//     Box 64 (AT5100-0100)/DRV Controlword/Controlword <-> Data Pointer/Control
//     Box 64 (AT5100-0100)/DRV Statusword/Statusword <-> Data Pointer/Status
//     Box 64 (AT5100-0100)/DRV Target torque/Target torque <-> Data Pointer/Torque
//     Box 64 (AT5100-0100)/DRV Torque actual value/Torque actual value <-> Data Pointer/ActTorque
//     Box 64 (AT5100-0100)/XFB Inputs/Data <-> Data Pointer/HallSensorValues
//   (this object) <-> TcCOM Objects/XTS ProcessingUnit 1/XL Part 2/XL Module 53
//     Box 65 (AT5100-0100)/DRV Commutation angle/Commutation angle <-> Data Pointer/CommutationAngle
//     Box 65 (AT5100-0100)/DRV Controlword/Controlword <-> Data Pointer/Control
//     Box 65 (AT5100-0100)/DRV Statusword/Statusword <-> Data Pointer/Status
//     Box 65 (AT5100-0100)/DRV Target torque/Target torque <-> Data Pointer/Torque
//     Box 65 (AT5100-0100)/DRV Torque actual value/Torque actual value <-> Data Pointer/ActTorque
//     Box 65 (AT5100-0100)/XFB Inputs/Data <-> Data Pointer/HallSensorValues
//   (this object) <-> TcCOM Objects/XTS ProcessingUnit 1/XL Part 2/XL Module 54
//     Box 66 (AT5100-0100)/DRV Commutation angle/Commutation angle <-> Data Pointer/CommutationAngle
//     Box 66 (AT5100-0100)/DRV Controlword/Controlword <-> Data Pointer/Control
//     Box 66 (AT5100-0100)/DRV Statusword/Statusword <-> Data Pointer/Status
//     Box 66 (AT5100-0100)/DRV Target torque/Target torque <-> Data Pointer/Torque
//     Box 66 (AT5100-0100)/DRV Torque actual value/Torque actual value <-> Data Pointer/ActTorque
//     Box 66 (AT5100-0100)/XFB Inputs/Data <-> Data Pointer/HallSensorValues
//   (this object) <-> TcCOM Objects/XTS ProcessingUnit 1/XL Part 2/XL Module 55
//     Box 67 (AT5100-0100)/DRV Commutation angle/Commutation angle <-> Data Pointer/CommutationAngle
//     Box 67 (AT5100-0100)/DRV Controlword/Controlword <-> Data Pointer/Control
//     Box 67 (AT5100-0100)/DRV Statusword/Statusword <-> Data Pointer/Status
//     Box 67 (AT5100-0100)/DRV Target torque/Target torque <-> Data Pointer/Torque
//     Box 67 (AT5100-0100)/DRV Torque actual value/Torque actual value <-> Data Pointer/ActTorque
//     Box 67 (AT5100-0100)/XFB Inputs/Data <-> Data Pointer/HallSensorValues
//   (this object) <-> TcCOM Objects/XTS ProcessingUnit 1/XL Part 2/XL Module 56
//     Box 68 (AT5100-0100)/DRV Commutation angle/Commutation angle <-> Data Pointer/CommutationAngle
//     Box 68 (AT5100-0100)/DRV Controlword/Controlword <-> Data Pointer/Control
//     Box 68 (AT5100-0100)/DRV Statusword/Statusword <-> Data Pointer/Status
//     Box 68 (AT5100-0100)/DRV Target torque/Target torque <-> Data Pointer/Torque
//     Box 68 (AT5100-0100)/DRV Torque actual value/Torque actual value <-> Data Pointer/ActTorque
//     Box 68 (AT5100-0100)/XFB Inputs/Data <-> Data Pointer/HallSensorValues
//   (this object) <-> TcCOM Objects/XTS ProcessingUnit 1/XL Part 2/XL Module 57
//     Box 69 (AT5100-0100)/DRV Commutation angle/Commutation angle <-> Data Pointer/CommutationAngle
//     Box 69 (AT5100-0100)/DRV Controlword/Controlword <-> Data Pointer/Control
//     Box 69 (AT5100-0100)/DRV Statusword/Statusword <-> Data Pointer/Status
//     Box 69 (AT5100-0100)/DRV Target torque/Target torque <-> Data Pointer/Torque
//     Box 69 (AT5100-0100)/DRV Torque actual value/Torque actual value <-> Data Pointer/ActTorque
//     Box 69 (AT5100-0100)/XFB Inputs/Data <-> Data Pointer/HallSensorValues
//   (this object) <-> TcCOM Objects/XTS ProcessingUnit 1/XL Part 3/XL Module 1
//     Box 74 (AT5100-0100)/DRV Commutation angle/Commutation angle <-> Data Pointer/CommutationAngle
//     Box 74 (AT5100-0100)/DRV Controlword/Controlword <-> Data Pointer/Control
//     Box 74 (AT5100-0100)/DRV Statusword/Statusword <-> Data Pointer/Status
//     Box 74 (AT5100-0100)/DRV Target torque/Target torque <-> Data Pointer/Torque
//     Box 74 (AT5100-0100)/DRV Torque actual value/Torque actual value <-> Data Pointer/ActTorque
//     Box 74 (AT5100-0100)/XFB Inputs/Data <-> Data Pointer/HallSensorValues
//   (this object) <-> TcCOM Objects/XTS ProcessingUnit 1/XL Part 3/XL Module 2
//     Box 75 (AT5100-0100)/DRV Commutation angle/Commutation angle <-> Data Pointer/CommutationAngle
//     Box 75 (AT5100-0100)/DRV Controlword/Controlword <-> Data Pointer/Control
//     Box 75 (AT5100-0100)/DRV Statusword/Statusword <-> Data Pointer/Status
//     Box 75 (AT5100-0100)/DRV Target torque/Target torque <-> Data Pointer/Torque
//     Box 75 (AT5100-0100)/DRV Torque actual value/Torque actual value <-> Data Pointer/ActTorque
//     Box 75 (AT5100-0100)/XFB Inputs/Data <-> Data Pointer/HallSensorValues
//   (this object) <-> TcCOM Objects/XTS ProcessingUnit 1/XL Part 3/XL Module 3
//     Box 76 (AT5100-0100)/DRV Commutation angle/Commutation angle <-> Data Pointer/CommutationAngle
//     Box 76 (AT5100-0100)/DRV Controlword/Controlword <-> Data Pointer/Control
//     Box 76 (AT5100-0100)/DRV Statusword/Statusword <-> Data Pointer/Status
//     Box 76 (AT5100-0100)/DRV Target torque/Target torque <-> Data Pointer/Torque
//     Box 76 (AT5100-0100)/DRV Torque actual value/Torque actual value <-> Data Pointer/ActTorque
//     Box 76 (AT5100-0100)/XFB Inputs/Data <-> Data Pointer/HallSensorValues
//   (this object) <-> TcCOM Objects/XTS ProcessingUnit 1/XL Part 3/XL Module 4
//     Box 77 (AT5100-0100)/DRV Commutation angle/Commutation angle <-> Data Pointer/CommutationAngle
//     Box 77 (AT5100-0100)/DRV Controlword/Controlword <-> Data Pointer/Control
//     Box 77 (AT5100-0100)/DRV Statusword/Statusword <-> Data Pointer/Status
//     Box 77 (AT5100-0100)/DRV Target torque/Target torque <-> Data Pointer/Torque
//     Box 77 (AT5100-0100)/DRV Torque actual value/Torque actual value <-> Data Pointer/ActTorque
//     Box 77 (AT5100-0100)/XFB Inputs/Data <-> Data Pointer/HallSensorValues
//   (this object) <-> TcCOM Objects/XTS ProcessingUnit 1/XL Part 3/XL Module 46
//     Box 72 (AT5100-0100)/DRV Commutation angle/Commutation angle <-> Data Pointer/CommutationAngle
//     Box 72 (AT5100-0100)/DRV Controlword/Controlword <-> Data Pointer/Control
//     Box 72 (AT5100-0100)/DRV Statusword/Statusword <-> Data Pointer/Status
//     Box 72 (AT5100-0100)/DRV Target torque/Target torque <-> Data Pointer/Torque
//     Box 72 (AT5100-0100)/DRV Torque actual value/Torque actual value <-> Data Pointer/ActTorque
//     Box 72 (AT5100-0100)/XFB Inputs/Data <-> Data Pointer/HallSensorValues
//   (this object) <-> TcCOM Objects/XTS ProcessingUnit 1/XL Part 3/XL Module 47
//     Box 73 (AT5100-0100)/DRV Commutation angle/Commutation angle <-> Data Pointer/CommutationAngle
//     Box 73 (AT5100-0100)/DRV Controlword/Controlword <-> Data Pointer/Control
//     Box 73 (AT5100-0100)/DRV Statusword/Statusword <-> Data Pointer/Status
//     Box 73 (AT5100-0100)/DRV Target torque/Target torque <-> Data Pointer/Torque
//     Box 73 (AT5100-0100)/DRV Torque actual value/Torque actual value <-> Data Pointer/ActTorque
//     Box 73 (AT5100-0100)/XFB Inputs/Data <-> Data Pointer/HallSensorValues
//   (this object) <-> TcCOM Objects/XTS ProcessingUnit 1/XL Part 3/XL Module 5
//     Box 78 (AT5100-0100)/DRV Commutation angle/Commutation angle <-> Data Pointer/CommutationAngle
//     Box 78 (AT5100-0100)/DRV Controlword/Controlword <-> Data Pointer/Control
//     Box 78 (AT5100-0100)/DRV Statusword/Statusword <-> Data Pointer/Status
//     Box 78 (AT5100-0100)/DRV Target torque/Target torque <-> Data Pointer/Torque
//     Box 78 (AT5100-0100)/DRV Torque actual value/Torque actual value <-> Data Pointer/ActTorque
//     Box 78 (AT5100-0100)/XFB Inputs/Data <-> Data Pointer/HallSensorValues
//   (this object) <-> TcCOM Objects/XTS ProcessingUnit 1/XL Part 3/XL Module 6
//     Box 79 (AT5100-0100)/DRV Commutation angle/Commutation angle <-> Data Pointer/CommutationAngle
//     Box 79 (AT5100-0100)/DRV Controlword/Controlword <-> Data Pointer/Control
//     Box 79 (AT5100-0100)/DRV Statusword/Statusword <-> Data Pointer/Status
//     Box 79 (AT5100-0100)/DRV Target torque/Target torque <-> Data Pointer/Torque
//     Box 79 (AT5100-0100)/DRV Torque actual value/Torque actual value <-> Data Pointer/ActTorque
//     Box 79 (AT5100-0100)/XFB Inputs/Data <-> Data Pointer/HallSensorValues
//   (this object) <-> TcCOM Objects/XTS ProcessingUnit 1/XL Part 3/XL Module 7
//     Box 80 (AT5100-0100)/DRV Commutation angle/Commutation angle <-> Data Pointer/CommutationAngle
//     Box 80 (AT5100-0100)/DRV Controlword/Controlword <-> Data Pointer/Control
//     Box 80 (AT5100-0100)/DRV Statusword/Statusword <-> Data Pointer/Status
//     Box 80 (AT5100-0100)/DRV Target torque/Target torque <-> Data Pointer/Torque
//     Box 80 (AT5100-0100)/DRV Torque actual value/Torque actual value <-> Data Pointer/ActTorque
//     Box 80 (AT5100-0100)/XFB Inputs/Data <-> Data Pointer/HallSensorValues
//   (this object) <-> TcCOM Objects/XTS ProcessingUnit 1/XL Part 3/XL Module 8
//     Box 81 (AT5100-0100)/DRV Commutation angle/Commutation angle <-> Data Pointer/CommutationAngle
//     Box 81 (AT5100-0100)/DRV Controlword/Controlword <-> Data Pointer/Control
//     Box 81 (AT5100-0100)/DRV Statusword/Statusword <-> Data Pointer/Status
//     Box 81 (AT5100-0100)/DRV Target torque/Target torque <-> Data Pointer/Torque
//     Box 81 (AT5100-0100)/DRV Torque actual value/Torque actual value <-> Data Pointer/ActTorque
//     Box 81 (AT5100-0100)/XFB Inputs/Data <-> Data Pointer/HallSensorValues

CONFIGURATION PlanarTrackMovement_1
    RESOURCE PLC ON TwinCAT3
        TASK PlcTask(INTERVAL := T#1ms, PRIORITY := 20);
        PROGRAM MAIN WITH PlcTask : MAIN;
    END_RESOURCE
END_CONFIGURATION

// ---- GVLs/GVL_General.TcGVL
VAR_GLOBAL CONSTANT

	nNumMaxMovers : UDINT :=16;
	nNumMaxTracks : UDINT :=3;
 	fMagnetEntry : LREAL := 8750; //PLEASE ENTER THE MAGNET ENTRY!!!
	fMagnetExit : LREAL := 9450; //PLEASE ENTER THE MAGNET EXIT!!!
END_VAR

VAR_GLOBAL
	aStopPositions : ARRAY [1..nNumMaxMovers] OF LREAL;// := [2400, 1700, 1000, 300];
	XtsOutterLoopOid: OTCID := 16#1010480;	
	XtsShortcutOid: OTCID := 16#1010490;
END_VAR

VAR_GLOBAL PERSISTENT
	nNumMovers: UDINT := 4;
END_VAR

// ---- POUs/MAIN.TcPOU
PROGRAM MAIN
VAR
		
	bAllDone		: BOOL;
	bStopSequence	: BOOL;
	
	nCase 		: INT;
	nMoveState		: ARRAY[1..nNumMaxMovers] OF INT;
	
	aDynamics	: ARRAY[1..nNumMaxMovers] OF DynamicConstraint_PathXY;
	aDynamicsFast	: ARRAY[1..nNumMaxMovers] OF DynamicConstraint_PathXY;
	aMoveOnTrackOptions : ARRAY[1..20] OF ST_MoveOnTrackOptions;
	
	fbXtsEnvironment: FB_TcIoXtsEnvironment;
	
	nForCounter: UDINT;
	M,N,T,Tr : UDINT;
	dynamics: INT;
	
	// Magnet
	MagnetValue AT%Q*: INT;
	bMagnetOn : BOOL;	
	stPositionInfo: ST_PositionInfo;
		
	pwm: FB_PWM;
	
	IsMoverCommandedInShortcut: BOOL;
	IsMoverInBlockingArea: BOOL;
	nActStopPos: UINT := 1;
	Fp_error : R_Trig;
	Velo : LREAL := 500;
	Switch : BOOL;
	WithoutSwitch : BOOL := TRUE;
	SwtichOnly: BOOL;
	
	MoverStop 	AT%I* :BOOL;
	MoverStopDone AT%Q*		: BOOL;
	Info 		AT%Q*: BOOL;
	Operating	AT%Q*: BOOL;
	Process		AT%Q*: BOOL;
	Fault		AT%Q*: BOOL;
	Emergency	AT%Q*: BOOL;
	
	Voltage1 AT%I*: UDINT;
	Voltage2 AT%I*: UDINT;
	
	
	TcRestart : TC_Restart;
	Restart : BOOL;
	busy : BOOL;
	fp_start : R_Trig;
	bStartSequence: BOOL;
	
	FP_Counter : r_trig;
	Switchcounter : DINT;
	SwitchCurrent: INT :=12000; 
	test : LREAL;
	Horntimer : tp; 
	R_trigHorn : R_trig;
	
	TestPowerMat : BOOL;
	StopPos : LREAL := 7611;
	StopTime : TIME := T#8S;
	StopTimer :ARRAY[1..nNumMaxMovers] OF ton;
	StartTimer :ARRAY[1..nNumMaxMovers] OF BOOL;
	
	
	MoverPos :ARRAY[1..nNumMaxMovers] OF PositionXYC;
	ArcLength :ARRAY[1..nNumMaxMovers] OF LREAL;
	TrackPos :ARRAY[1..nNumMaxMovers] OF ARRAY[1..nNumMaxTracks] OF PositionXYC;
	
	GetMoverOnTrack : ReadTcCom;
	aMoverTrack : ARRAY[1..nNumMaxMovers] OF otcid;
	FirstMoverTrackPos : LREAL;
	MoverGap : LREAL;
	FTrigTrackCount : F_Trig;
	MoverNo  : UDINT;
END_VAR

fbXtsEnvironment.Init(TRUE);

Emergency :=  MoverStop;

Operating := NOT  MoverStop;
R_trigHorn(clk := Voltage1> 10000 OR Voltage2 >10000);
Horntimer(in:= ( R_trigHorn.Q ) , PT:= T#2S,Q=> info);

IF nCASE > 90 THEN
	Process := TRUE;
ELSE 
	Process := FALSE;	
END_IF





IF NOT fbXtsEnvironment.P_IsInitialized THEN
	RETURN;
END_IF





IF GetMoverOnTrack.GetComObject(MC_Tracks[1].MCTOPLC_STD.TrackOID)THEN
	aMoverTrack:= GetMoverOnTrack.GetValue();
END_IF







IF NOT MoverStop AND NOT MoverStopDone THEN
	FOR nForCounter:=1 TO nNumMovers DO
		aDynamics[nForCounter].SetValuesVADJ(8000, 8000, 8000, 20000);
		nCase := 140;
		//fbPlanarMover[nForCounter].McPlanarMover.Halt(MoverFeedback[nForCounter], aDynamics[nForCounter]);
	END_FOR		
	MoverStopDone := TRUE;
ELSIF 	MoverStop THEN
	MoverStopDone := FALSE;
END_IF


	TcRestart(
	NETID:= '', 
	RESTART:= Restart, 
	TMOUT:=T#5S , 
	BUSY=>busy , 
	ERR=> , 
	ERRID=> );


fp_start(clk:=bStartSequence);
IF fp_start.Q THEN
	nCase := 10;
	bStartSequence := FALSE;
END_IF



IsMoverInBlockingArea := FALSE;
FOR M := 1 TO nNumMovers DO///Movers
	StopTimer[M](in:=StartTimer[m],PT:=StopTime);
	fbPlanarMover[m].nMoverId := nForCounter;
	fbPlanarMover[m].iTcIoXtsXpuMover := fbXtsEnvironment.XpuTcIo(1).MoverTcIo(TO_UINT(m));
	fbPlanarMover[m].Update();
	
	GVL_mc3.Mover[M].MoverPos  :=fbPlanarMover[M].McPlanarMover.MCTOPLC.SETONTRACK.SetPos;
	GVL_mc3.Mover[M].TrackID:= fbPlanarMover[M].McPlanarMover.MCTOPLC.SETONTRACK.TrackOID;
	GVL_mc3.Mover[M].MoverNumber := M;
	
	MoverPos[M].SetValuesXYC(fbPlanarMover[M].McPlanarMover.MCTOPLC.SET.SetPos.x ,fbPlanarMover[M].McPlanarMover.MCTOPLC.SET.SetPos.y,fbPlanarMover[M].McPlanarMover.MCTOPLC.SET.SetPos.c);
	
	TR := Tr+1;
	IF Tr = 4 THEN
		Tr :=1;
	END_IF
	ArcLength[M] :=GVL_Mc3.MC_Tracks[Tr].GetArcLengthClosestTo(MoverPos[M]);
	GVL_Mc3.MC_Tracks[Tr].GetPositionAt(ArcLength[M],TrackPos[M][Tr]);
	
	IF ABS(MoverPos[m].x - TrackPos[M][Tr].x) < 1 AND  ABS(MoverPos[m].y - TrackPos[M][Tr].y) < 1 THEN
 		GVL_mc3.Mover[M].MoverTrackNr := Tr;
	END_IF	
	
	

	IsMoverInBlockingArea := IsMoverInBlockingArea OR (Mover[M].TrackID = GVL_Mc3.MC_Tracks[E_TrackNum.main].MCTOPLC_STD.TrackOID AND IsBetween(Mover[M].MoverPos, fMagnetEntry - 100, fMagnetExit + 100));
	MoverFeedback[M].Update();
//	Fp_error(clk := fbPlanarMover[M].McPlanarMover.Error);
	IF Fp_error.Q THEN
		nCase := 140;
		Fault := TRUE;
		bMagnetOn := FALSE;
	ELSE
		Fault := FALSE;
	END_IF
	
	IF aMoverTrack[1] <> 0 AND_THEN fbPlanarMover[m].McPlanarMover.MCTOPLC.STD.MoverOID = aMoverTrack[1] THEN
		FirstMoverTrackPos := fbPlanarMover[m].McPlanarMover.MCTOPLC.SETONTRACK.SetPos;
	END_IF
	
	

	
	
END_FOR

FOR T := 1 TO nNumMaxTracks DO 
	MC_Tracks[T].Update();
	MC_Trackfeedback[T].Update();
	
END_FOR
 MoverGap := (GVL_Mc3.MC_Tracks[E_TrackNum.Big].GetLength()- FirstMoverTrackPos);
(*
FTrigTrackCount(CLK:=GVL_Mc3.MC_Tracks[E_TrackNum.Small].MCTOPLC_STD.MoverCountOnTrack =0);
IF FTrigTrackCount.Q    THEN
	IsMoverCommandedInShortcut := FALSE;
END_IF	
*)

CASE nCase OF
	10:
		FOR nForCounter := 1 TO fbXtsEnvironment.XpuTcIo(1).GetPartCount() DO
			fbXtsEnvironment.XpuTcIo(1).PartTcIo(TO_UINT(nForCounter)).TriggerReset();
		END_FOR
		Fault := FALSE;
		nCase := 20;

	20:
		FOR T := 1 TO nNumMaxTracks DO 
			MC_Tracks[T].Enable(MC_Trackfeedback[T]);
		END_FOR
				nCase := 30;
		
		
	30: 
		IF MC_Trackfeedback[1].Done AND MC_Trackfeedback[2].Done AND MC_Trackfeedback[3].Done THEN
			nCase := 35;
		END_IF
		
		
	35:
		FOR nForCounter:=1 TO nNumMovers DO
			fbPlanarMover[nForCounter].McPlanarMover.Reset(MoverFeedback[nForCounter]);
		END_FOR
		nCase := 36;	
		
		
	36:	
		bAllDone:=TRUE;
		FOR nForCounter:=1 TO nNumMovers DO
			bAllDone:=bAllDone AND MoverFeedback[nForCounter].Done;
		END_FOR
		
		IF bAllDone THEN
			nCase := 40;
		END_IF
		
		
	40:
		FOR nForCounter:=1 TO nNumMovers DO
			fbPlanarMover[nForCounter].McPlanarMover.Enable(MoverFeedback[nForCounter]);
		END_FOR
		nCase := 50;
	
		
	50:
		bAllDone:=TRUE;
		FOR nForCounter:=1 TO nNumMovers DO
			bAllDone:=bAllDone AND MoverFeedback[nForCounter].Done;
		END_FOR
		
		IF bAllDone THEN
			nCase := 60;
		END_IF

	//55:

	60:
		FOR nForCounter:=nNumMovers TO 1  BY -1 DO
			fbPlanarMover[nForCounter].JoinTrack(MoverFeedback[nForCounter], GVL_Mc3.MC_Tracks[3]);//  Mover[nForCounter].MoverTrackNr]);//
		END_FOR
		
		nCase := 70;
		
		
	70:
		bAllDone:=TRUE;
		FOR nForCounter:=1 TO nNumMovers DO
			bAllDone:=bAllDone AND MoverFeedback[nForCounter].Done;
		END_FOR
		
		IF bAllDone THEN
			nCase := 80;
		END_IF
		
	80:	
		FOR nForCounter:=1 TO nNumMovers DO
			nMoveState[nForCounter] := 0;
			aMoveOnTrackOptions[nForCounter].direction := MC_Direction.mcDirectionPositive;
			aMoveOnTrackOptions[nForCounter].gapMode := MC_GAP_MODE_ON_TRACK.Fast1D;
		END_FOR
		
		nCase := 90;

	100:
		
		FOR nForCounter:=1 TO nNumMovers DO
			aDynamicsFast[nForCounter].SetValuesVADJ(Velo, 16000, 16000, 29000);
			aDynamics[nForCounter].SetValuesVADJ(Velo, 10000, 1500, 29000);
			aMoveOnTrackOptions[nForCounter].gap:= 800;//900;	 
		END_FOR
	aDynamics[1].SetValuesVADJ(Velo-test,  30000, 1000, 10000);
		FOR nForCounter:=1 TO nNumMovers DO
	
			
			IF MoverNo <> 0 AND_THEN 	fbPlanarMover[MoverNo].McPlanarMover.MCTOPLC.SETONTRACK.TrackOID =	 GVL_Mc3.MC_Tracks[E_TrackNum.Big].MCTOPLC_STD.TrackOID THEN
				IsMoverCommandedInShortcut := FALSE;
			//	MoverNo := 0;
			END_IF
				
			CASE nMoveState[nForCounter] OF
				
				0: // Track 3 Main Cycel 
					fbPlanarMover[nForCounter].McPlanarMover.MoveOnTrack(MoverFeedback[nForCounter], GVL_Mc3.MC_Tracks[E_TrackNum.Main],  GVL_Mc3.MC_Tracks[E_TrackNum.Main].GetLength()-500, aDynamics[nForCounter], aMoveOnTrackOptions[nForCounter]);
					nMoveState[nForCounter] := 10;
					
				10:
					IF Mover[nForCounter].MoverPos > GVL_Mc3.MC_Tracks[E_TrackNum.Main].GetLength()-6000  AND  Mover[nForCounter].TrackID =   GVL_Mc3.MC_Tracks[E_TrackNum.Main].MCTOPLC_STD.TrackOID    THEN//     MCTrackOid_MainSemicircle THEN
						IF  (SwtichOnly OR NOT IsMoverCommandedInShortcut )AND NOT WithoutSwitch  AND  nForCounter > 10 THEN
							nMoveState[nForCounter] := 40; // 20 - BigCycel
							//IF fbPlanarMover[nForCounter].IsCommandedInShortcut THEN
								IsMoverCommandedInShortcut := TRUE;
								MoverNo :=nForCounter; /// fbPlanarMover[nForCounter].McPlanarMover.MCTOPLC.STD.MoverOID;
							//END_IF
						ELSE
							nMoveState[nForCounter] := 20;  // 40- SmallCycel					
						END_IF
					END_IF

				
				20:
					fbPlanarMover[nForCounter].McPlanarMover.MoveOnTrack(MoverFeedback[nForCounter], GVL_Mc3.MC_Tracks[E_TrackNum.Big], GVL_Mc3.MC_Tracks[E_TrackNum.Big].GetLength()-2000, aDynamics[nForCounter],aMoveOnTrackOptions[nForCounter]);
					nMoveState[nForCounter] := 30;
				
					
				30:
					IF Mover[nForCounter].MoverPos > GVL_Mc3.MC_Tracks[E_TrackNum.Big].GetLength()-4000 AND  Mover[nForCounter].TrackID = GVL_Mc3.MC_Tracks[E_TrackNum.big].MCTOPLC_STD.TrackOID    THEN//      MCTrackOid_BigSemicircle THEN
						nMoveState[nForCounter] := 0;
					END_IF				
				
			
				40:
					fbPlanarMover[nForCounter].McPlanarMover.MoveOnTrack(MoverFeedback[nForCounter], GVL_Mc3.MC_Tracks[E_TrackNum.Small], (GVL_Mc3.MC_Tracks[E_TrackNum.Small].GetLength()-3000), aDynamics[nForCounter], aMoveOnTrackOptions[nForCounter]);
					nMoveState[nForCounter] := 50;	

			

			
				50:
					IF Mover[nForCounter].MoverPos > GVL_Mc3.MC_Tracks[E_TrackNum.small].GetLength()-3500 AND  Mover[nForCounter].TrackID = GVL_Mc3.MC_Tracks[E_TrackNum.Small].MCTOPLC_STD.TrackOID    THEN// MCTrackOid_Shortcut THEN
						nMoveState[nForCounter] := 60;
					END_IF
				60:
					 // Track 3 Main Cycel
					IF FirstMoverTrackPos > 800 THEN 
						fbPlanarMover[nForCounter].McPlanarMover.MoveOnTrack(MoverFeedback[nForCounter], GVL_Mc3.MC_Tracks[E_TrackNum.Main],  GVL_Mc3.MC_Tracks[E_TrackNum.Main].GetLength()-500, aDynamicsFast[nForCounter], aMoveOnTrackOptions[nForCounter]);
						nMoveState[nForCounter] := 10;
					END_IF
				END_CASE
		
		END_FOR

		IF bStopSequence AND NOT(IsMoverInBlockingArea) THEN
			nCase := 110;
			bStopSequence := FALSE;
		END_IF
		110:
			N:= nNumMovers;
			FOR nForCounter:=1 TO nNumMovers DO		
				GVL_General.aStopPositions[nForCounter] := TO_LREAL(  fbXtsEnvironment.XpuTcIo(1).MoverTcIo(TO_UINT(N)).GetSimulatedStartUpPosition());
				N := N -1;
			END_FOR
			nCase := 120;
		
		120:	
			nActStopPos := UDINT_TO_UINT(nNumMaxMovers-nNumMovers+1);
			FOR nForCounter:=1 TO nNumMovers DO
				aDynamics[nForCounter].SetValuesVADJ(1000, 4000, 4000, 10000);
				nMoveState[nForCounter] := 0;
				fbPlanarMover[nForCounter].McPlanarMover.MoveOnTrack(MoverFeedback[nForCounter], GVL_Mc3.MC_Tracks[E_TrackNum.main], 300, aDynamics[nForCounter],aMoveOnTrackOptions[nForCounter]);
			END_FOR

			nCase:= 130; 
		130:
			FOR nForCounter:=1 TO nNumMaxMovers - (nNumMaxMovers -nNumMovers)  DO
				CASE nMoveState[nForCounter] OF
					0:								
						
						IF Mover[nForCounter].MoverPos < 300 AND  Mover[nForCounter].TrackID = GVL_Mc3.MC_Tracks[E_TrackNum.main].MCTOPLC_STD.TrackOID THEN
							aMoveOnTrackOptions[nForCounter].gap:= 700;
							fbPlanarMover[nForCounter].McPlanarMover.MoveOnTrack(MoverFeedback[nForCounter], GVL_Mc3.MC_Tracks[E_TrackNum.main], aStopPositions[nActStopPos], aDynamics[nForCounter], aMoveOnTrackOptions[nForCounter]);
							nActStopPos := nActStopPos + 1;
							nMoveState[nForCounter] := 10;
						END_IF
				END_CASE
			END_FOR
		
			bAllDone := TRUE;
			FOR nForCounter:=1 TO nNumMovers DO
				IF NOT(MoverFeedback[nForCounter].Done OR MoverFeedback[nForCounter].Error) THEN
					bAllDone := FALSE;
					EXIT;
				END_IF
			END_FOR
			
			IF bAllDone THEN
				nCase := 150;
			END_IF
		
		140:
			FOR nForCounter:=1 TO nNumMovers DO
				fbPlanarMover[nForCounter].McPlanarMover.Halt(MoverFeedback[nForCounter], aDynamics[nForCounter]);
			END_FOR	
			
			nCase := 145;
			
		145:
			bAllDone := TRUE;
			FOR nForCounter:=1 TO nNumMovers DO
				IF NOT(MoverFeedback[nForCounter].Done OR MoverFeedback[nForCounter].Error) THEN
					bAllDone := FALSE;
					EXIT;
				END_IF
			END_FOR
			
			IF bAllDone THEN
				nCase := 150;
			END_IF
		
		//Disable
		150:
			MoverStopDone := TRUE;
			FOR nForCounter:=1 TO nNumMovers DO
				fbPlanarMover[nForCounter].McPlanarMover.Disable(MoverFeedback[nForCounter]);
			END_FOR
				
			nCase := 0;
END_CASE

bMagnetOn := FALSE;
FOR nForCounter:=1 TO nNumMovers DO
	stPositionInfo := fbXtsEnvironment.XpuTcIo(1).MoverTcIo(TO_UINT(nForCounter)).GetPositionInfo();
	IF stPositionInfo.nTrackObjectId = XtsShortcutOid AND (IsBetween(stPositionInfo.fTrackPosition, fMagnetEntry - (Velo*0.08), fMagnetExit)) THEN
		bMagnetOn := TRUE;
	END_IF
END_FOR

pwm();
	
IF bMagnetOn AND NOT Fault THEN
	MagnetValue := SwitchCurrent*1310;
ELSE
 	MagnetValue := 0;
END_IF

FP_Counter(clk:=bMagnetOn);

IF FP_Counter.Q THEN
	Switchcounter := Switchcounter+1;

END_IF

END_PROGRAM

// ---- POUs/ReadTcCom.TcPOU
FUNCTION_BLOCK ReadTcCom
VAR_INPUT
	
END_VAR
VAR_OUTPUT
	bBusy 				: BOOL;
	bDone 				: BOOL;
	bError 				: BOOL;
	bGetComObject	: BOOL;
END_VAR
VAR
	
	_nObjectId				: OTCID;
	_ipComObject 			: ITComObject;
	_nSoftDriveOid			: OTCID;
	PID_Value	: PTCID := 	16#05030149;
END_VAR

METHOD GetComObject : BOOL
VAR_INPUT
	nObjectId	: OTCID;
END_VAR
IF FW_ObjMgr_GetObjectInstance(	oid		:= nObjectId, 
								iid		:= TC_GLOBAL_IID_LIST.IID_ITComObject, 
								pipUnk	:= ADR(_ipComObject)) = 0
THEN
	GetComObject := TRUE;
END_IF
END_METHOD

METHOD GetValue : ARRAY[1..nNumMaxMovers] OF OTCID
VAR_INPUT
	//PID_Value 		: otcid;
END_VAR
VAR
	Value			: ARRAY[1..nNumMaxMovers] OF OTCID;
	nData 			: UDINT := SIZEOF(Value);
	pData 			: PVOID := ADR(Value);
	stEventEntry	: TcEventEntry;
	pstEventEntry	: REFERENCE TO TcEventEntry REF= stEventEntry;
	
END_VAR
VAR_INST
	hResult : HRESULT;
END_VAR
IF _ipComObject <> 0  THEN
	 hResult := _ipComObject.TcGetObjPara(
				pid 	:= PID_Value,
				nData 	:= nData,
				pData 	:= pData,
				pgp   	:=0) ;
	IF hResult = 0	THEN
		GetValue := Value;
		bError := FALSE;
	ELSE
		bError := TRUE;
	END_IF
END_IF
END_METHOD

END_FUNCTION_BLOCK

// ---- POUs/IsBetween.TcPOU
FUNCTION IsBetween : BOOL
VAR_INPUT
	value: 	LREAL;
	minV:	LREAL;
	maxV:	LREAL;
END_VAR
VAR
END_VAR

IsBetween := value > minV AND value < maxV;

END_FUNCTION

// ---- POUs/FB_PlanarMover.TcPOU
FUNCTION_BLOCK FB_PlanarMover

VAR_INPUT
	nMoverId			: UDINT;
	iTcIoXtsXpuMover	: I_TcIoXtsXpuMover;
END_VAR

VAR
	_McPlanarMover	: MC_PlanarMover;
	_PlanarTrail    : MC_PlanarTrackTrail;
  	

END_VAR

PROPERTY IsCommandedInShortcut : BOOL
GET
VAR
	nCounter: UDINT := 0;
END_VAR
_mcPlanarMover.GetTrackTrailInformation(_PlanarTrail);

IF  _PlanarTrail.Size > 1 THEN
	FOR nCounter := 1 TO _PlanarTrail.Size  DO
		IF _PlanarTrail.GetTrackOidAt(nCounter) = GVL_Mc3.MC_Tracks[E_Tracknum.Small].MCTOPLC_STD.TrackOID  THEN
			IsCommandedInShortcut := TRUE;
		END_IF
	END_FOR
END_IF
END_GET
SET
END_SET
END_PROPERTY

METHOD JoinTrack

VAR_INPUT
	feedback: REFERENCE TO MC_PlanarFeedback;
END_VAR

VAR_IN_OUT
	track: MC_PlanarTrack;
END_VAR
_McPlanarMover.JoinTrack(feedback, track, 0, 0);
END_METHOD

PROPERTY McPlanarMover : REFERENCE TO MC_PlanarMover
GET
McPlanarMover ref= _McPlanarMover;
END_GET
END_PROPERTY

METHOD Update : PVOID
_mcPlanarMover.Update();


_mcPlanarMover.GetTrackTrailInformation(_PlanarTrail);

IF(* _PlanarTrail.Error OR*) _PlanarTrail.Size < 1 THEN
   RETURN;
END_IF
   
//SmallCircle
IF _PlanarTrail.GetTrackOidAt(2) = MC_Tracks[E_TrackNum.Small].MCTOPLC_STD.TrackOID   THEN
	iTcIoXtsXpuMover.SetActiveTrackObjectId(XtsShortcutOid);
//BigCircle
ELSIF _PlanarTrail.GetTrackOidAt(2) =MC_Tracks[E_TrackNum.Big].MCTOPLC_STD.TrackOID THEN
	iTcIoXtsXpuMover.SetActiveTrackObjectId(XtsOutterLoopOid);
END_IF
END_METHOD

END_FUNCTION_BLOCK
